// TIA Portal V17 export
// export: Created 2025-04-25T10:06:56.2061838Z, ExportSetting WithDefaults, DisplayName Totally Integrated Automation Portal, DisplayVersion V17 Update 8, DisplayName TIA Portal Openness, DisplayVersion V17 Update 8, DisplayName TIA Portal Version Control Interface, DisplayVersion V17, DisplayName SINAMICS Startdrive Advanced, DisplayVersion V17 SP2, DisplayName SINAMICS Startdrive G110M, G120, G120C, G120D, G120P, G115D, DisplayVersion V17 SP2, DisplayName SINAMICS Startdrive G130, G150, S120, S150, SINAMICS MV, S210, DisplayVersion V17 SP2, DisplayName STEP 7 Professional, DisplayVersion V17 Update 8, DisplayName SINUMERIK ONE STEP 7 Toolbox, DisplayVersion V17 Update 12, DisplayName SINUMERIK 840D sl STEP 7 Toolbox, DisplayVersion V17 Update 12, DisplayName STEP 7 Safety, DisplayVersion V17 Update 6, DisplayName WinCC Advanced / Unified PC, DisplayVersion V17 Update 8
FUNCTION "FC2810_U1_F4_GRIPPER" : Void   // FC2810, LAD
TITLE = FC2810_F4_GRIPPER
{ S7_Optimized_Access := 'FALSE' }
AUTHOR : ETXETAR
VERSION : 1.0
// stored: AutoNumber false, IsIECCheckEnabled false, SetENOAutomatically false, UDAEnableTagReadback false
   VAR_TEMP
      RET_VAL_1 : Int;
      UNIT_NUMBER : UInt;
      STATION_NUMBER : UInt;
   END_VAR
BEGIN

REGION Network 1: CALL FB2509 FIXTURE 1 GRIPPER
   // 2#0000_0001 OPTIONS 0 BIT 0 LOCATED INPUT 1 OPTION
   // 2#0000_0010 OPTIONS 0 BIT 1 LOCATED INPUT 2 OPTION
   // 2#0000_0100 OPTIONS 0 BIT 2 LOCATED INPUT 3 OPTION
   // 2#0000_1000 OPTIONS 0 BIT 3 LOCATED INPUT 4 OPTION
   // 2#0001_0000 OPTIONS 0 BIT 4 LOCATED PRESSURE INPUT 1 OPTION
   // 2#0010_0000 OPTIONS 0 BIT 5 LOCATED PRESSURE INPUT 2 OPTION
   // 2#0100_0000 OPTIONS 0 BIT 6 LOW PRESSURE INPUT 1 OPTION
   // 2#1000_0000 OPTIONS 0 BIT 7 SPARE OPTION
   // 
   // 2#0000_0001 OPTIONS 1 BIT 0 RETURNED INPUT 1 OPTION
   // 2#0000_0010 OPTIONS 1 BIT 1 RETURNED INPUT 2 OPTION
   // 2#0000_0100 OPTIONS 1 BIT 2 RETURNED INPUT 3 OPTION
   // 2#0000_1000 OPTIONS 1 BIT 3 RETURNED INPUT 4 OPTION
   // 2#0001_0000 OPTIONS 1 BIT 4 RETURNED PRESSURE INPUT 1 OPTION
   // 2#0010_0000 OPTIONS 1 BIT 5 RETURNED PRESSURE INPUT 2 OPTION
   // 2#0100_0000 OPTIONS 1 BIT 6 SPARE OPTION
   // 2#1000_0000 OPTIONS 1 BIT 7 SPARE OPTION
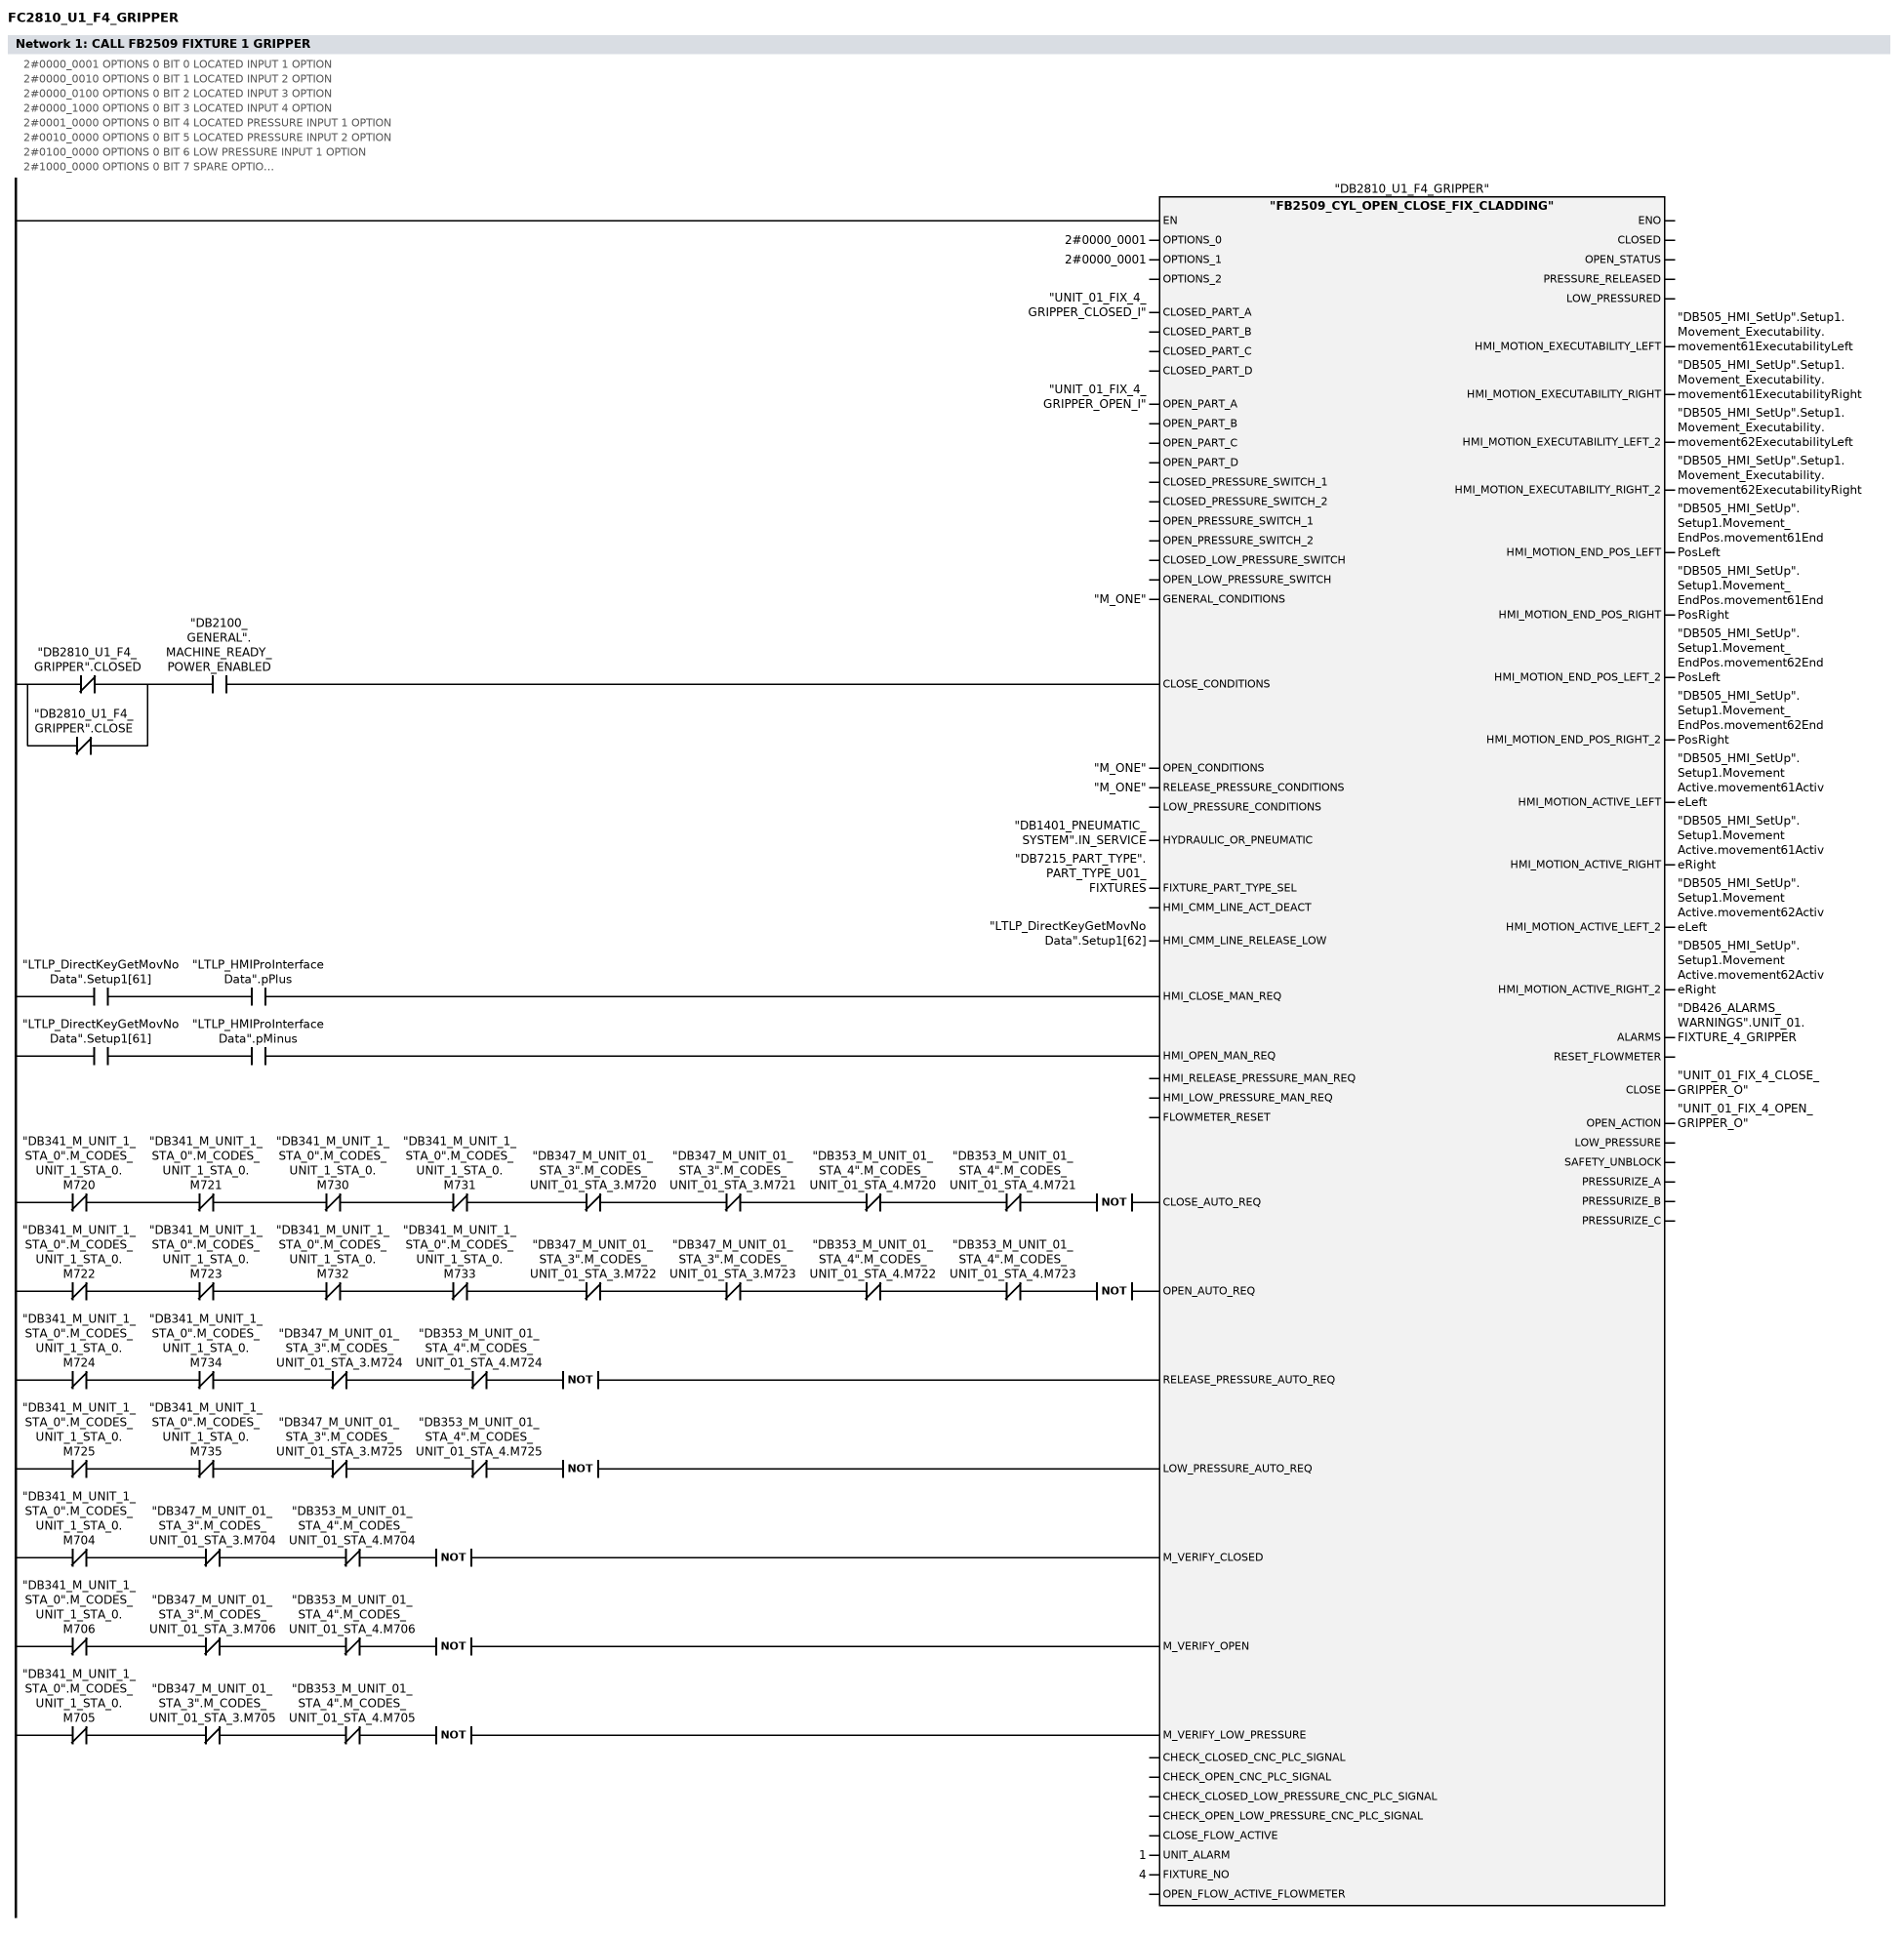
   RUNG wire#powerrail
      "DB2810_U1_F4_GRIPPER"(CLOSE_CONDITIONS := wire#w2, HMI_CLOSE_MAN_REQ := wire#w3, HMI_OPEN_MAN_REQ := wire#w4, CLOSE_AUTO_REQ := wire#w5, OPEN_AUTO_REQ := wire#w6, RELEASE_PRESSURE_AUTO_REQ := wire#w7, LOW_PRESSURE_AUTO_REQ := wire#w8, M_VERIFY_CLOSED := wire#w9, M_VERIFY_OPEN := wire#w10, M_VERIFY_LOW_PRESSURE := wire#w11, OPTIONS_0 := 2#0000_0001, OPTIONS_1 := 2#0000_0001, OPTIONS_2 :=, CLOSED_PART_A := "UNIT_01_FIX_4_GRIPPER_CLOSED_I", CLOSED_PART_B :=, CLOSED_PART_C :=, CLOSED_PART_D :=, OPEN_PART_A := "UNIT_01_FIX_4_GRIPPER_OPEN_I", OPEN_PART_B :=, OPEN_PART_C :=, OPEN_PART_D :=, CLOSED_PRESSURE_SWITCH_1 :=, CLOSED_PRESSURE_SWITCH_2 :=, OPEN_PRESSURE_SWITCH_1 :=, OPEN_PRESSURE_SWITCH_2 :=, CLOSED_LOW_PRESSURE_SWITCH :=, OPEN_LOW_PRESSURE_SWITCH :=, GENERAL_CONDITIONS := "M_ONE", OPEN_CONDITIONS := "M_ONE", RELEASE_PRESSURE_CONDITIONS := "M_ONE", LOW_PRESSURE_CONDITIONS :=, HYDRAULIC_OR_PNEUMATIC := "DB1401_PNEUMATIC_SYSTEM".IN_SERVICE, FIXTURE_PART_TYPE_SEL := "DB7215_PART_TYPE".PART_TYPE_U01_FIXTURES, HMI_CMM_LINE_ACT_DEACT :=, HMI_CMM_LINE_RELEASE_LOW := "LTLP_DirectKeyGetMovNoData".Setup1[62], HMI_RELEASE_PRESSURE_MAN_REQ :=, HMI_LOW_PRESSURE_MAN_REQ :=, FLOWMETER_RESET :=, CHECK_CLOSED_CNC_PLC_SIGNAL :=, CHECK_OPEN_CNC_PLC_SIGNAL :=, CHECK_CLOSED_LOW_PRESSURE_CNC_PLC_SIGNAL :=, CHECK_OPEN_LOW_PRESSURE_CNC_PLC_SIGNAL :=, CLOSE_FLOW_ACTIVE :=, UNIT_ALARM := 1, FIXTURE_NO := 4, OPEN_FLOW_ACTIVE_FLOWMETER :=, CLOSED =>, OPEN_STATUS =>, PRESSURE_RELEASED =>, LOW_PRESSURED =>, HMI_MOTION_EXECUTABILITY_LEFT => "DB505_HMI_SetUp".Setup1.Movement_Executability.movement61ExecutabilityLeft, HMI_MOTION_EXECUTABILITY_RIGHT => "DB505_HMI_SetUp".Setup1.Movement_Executability.movement61ExecutabilityRight, HMI_MOTION_EXECUTABILITY_LEFT_2 => "DB505_HMI_SetUp".Setup1.Movement_Executability.movement62ExecutabilityLeft, HMI_MOTION_EXECUTABILITY_RIGHT_2 => "DB505_HMI_SetUp".Setup1.Movement_Executability.movement62ExecutabilityRight, HMI_MOTION_END_POS_LEFT => "DB505_HMI_SetUp".Setup1.Movement_EndPos.movement61EndPosLeft, HMI_MOTION_END_POS_RIGHT => "DB505_HMI_SetUp".Setup1.Movement_EndPos.movement61EndPosRight, HMI_MOTION_END_POS_LEFT_2 => "DB505_HMI_SetUp".Setup1.Movement_EndPos.movement62EndPosLeft, HMI_MOTION_END_POS_RIGHT_2 => "DB505_HMI_SetUp".Setup1.Movement_EndPos.movement62EndPosRight, HMI_MOTION_ACTIVE_LEFT => "DB505_HMI_SetUp".Setup1.MovementActive.movement61ActiveLeft, HMI_MOTION_ACTIVE_RIGHT => "DB505_HMI_SetUp".Setup1.MovementActive.movement61ActiveRight, HMI_MOTION_ACTIVE_LEFT_2 => "DB505_HMI_SetUp".Setup1.MovementActive.movement62ActiveLeft, HMI_MOTION_ACTIVE_RIGHT_2 => "DB505_HMI_SetUp".Setup1.MovementActive.movement62ActiveRight, ALARMS => "DB426_ALARMS_WARNINGS".UNIT_01.FIXTURE_4_GRIPPER, RESET_FLOWMETER =>, CLOSE => "UNIT_01_FIX_4_CLOSE_GRIPPER_O", OPEN_ACTION => "UNIT_01_FIX_4_OPEN_GRIPPER_O", LOW_PRESSURE =>, SAFETY_UNBLOCK =>, PRESSURIZE_A =>, PRESSURIZE_B =>, PRESSURIZE_C =>)
   END_RUNG
   RUNG wire#powerrail
      I_Contact( "DB2810_U1_F4_GRIPPER".CLOSED )
      wire#w1
      Contact( "DB2100_GENERAL".MACHINE_READY_POWER_ENABLED )
   END_RUNG wire#w2
   RUNG wire#powerrail
      I_Contact( "DB2810_U1_F4_GRIPPER".CLOSE )
   END_RUNG wire#w1
   RUNG wire#powerrail
      Contact( "LTLP_DirectKeyGetMovNoData".Setup1[61] )
      Contact( "LTLP_HMIProInterfaceData".pPlus )
   END_RUNG wire#w3
   RUNG wire#powerrail
      Contact( "LTLP_DirectKeyGetMovNoData".Setup1[61] )
      Contact( "LTLP_HMIProInterfaceData".pMinus )
   END_RUNG wire#w4
   RUNG wire#powerrail
      I_Contact( "DB341_M_UNIT_1_STA_0".M_CODES_UNIT_1_STA_0.M720 )
      I_Contact( "DB341_M_UNIT_1_STA_0".M_CODES_UNIT_1_STA_0.M721 )
      I_Contact( "DB341_M_UNIT_1_STA_0".M_CODES_UNIT_1_STA_0.M730 )
      I_Contact( "DB341_M_UNIT_1_STA_0".M_CODES_UNIT_1_STA_0.M731 )
      I_Contact( "DB347_M_UNIT_01_STA_3".M_CODES_UNIT_01_STA_3.M720 )
      I_Contact( "DB347_M_UNIT_01_STA_3".M_CODES_UNIT_01_STA_3.M721 )
      I_Contact( "DB353_M_UNIT_01_STA_4".M_CODES_UNIT_01_STA_4.M720 )
      I_Contact( "DB353_M_UNIT_01_STA_4".M_CODES_UNIT_01_STA_4.M721 )
      Not()
   END_RUNG wire#w5
   RUNG wire#powerrail
      I_Contact( "DB341_M_UNIT_1_STA_0".M_CODES_UNIT_1_STA_0.M722 )
      I_Contact( "DB341_M_UNIT_1_STA_0".M_CODES_UNIT_1_STA_0.M723 )
      I_Contact( "DB341_M_UNIT_1_STA_0".M_CODES_UNIT_1_STA_0.M732 )
      I_Contact( "DB341_M_UNIT_1_STA_0".M_CODES_UNIT_1_STA_0.M733 )
      I_Contact( "DB347_M_UNIT_01_STA_3".M_CODES_UNIT_01_STA_3.M722 )
      I_Contact( "DB347_M_UNIT_01_STA_3".M_CODES_UNIT_01_STA_3.M723 )
      I_Contact( "DB353_M_UNIT_01_STA_4".M_CODES_UNIT_01_STA_4.M722 )
      I_Contact( "DB353_M_UNIT_01_STA_4".M_CODES_UNIT_01_STA_4.M723 )
      Not()
   END_RUNG wire#w6
   RUNG wire#powerrail
      I_Contact( "DB341_M_UNIT_1_STA_0".M_CODES_UNIT_1_STA_0.M724 )
      I_Contact( "DB341_M_UNIT_1_STA_0".M_CODES_UNIT_1_STA_0.M734 )
      I_Contact( "DB347_M_UNIT_01_STA_3".M_CODES_UNIT_01_STA_3.M724 )
      I_Contact( "DB353_M_UNIT_01_STA_4".M_CODES_UNIT_01_STA_4.M724 )
      Not()
   END_RUNG wire#w7
   RUNG wire#powerrail
      I_Contact( "DB341_M_UNIT_1_STA_0".M_CODES_UNIT_1_STA_0.M725 )
      I_Contact( "DB341_M_UNIT_1_STA_0".M_CODES_UNIT_1_STA_0.M735 )
      I_Contact( "DB347_M_UNIT_01_STA_3".M_CODES_UNIT_01_STA_3.M725 )
      I_Contact( "DB353_M_UNIT_01_STA_4".M_CODES_UNIT_01_STA_4.M725 )
      Not()
   END_RUNG wire#w8
   RUNG wire#powerrail
      I_Contact( "DB341_M_UNIT_1_STA_0".M_CODES_UNIT_1_STA_0.M704 )
      I_Contact( "DB347_M_UNIT_01_STA_3".M_CODES_UNIT_01_STA_3.M704 )
      I_Contact( "DB353_M_UNIT_01_STA_4".M_CODES_UNIT_01_STA_4.M704 )
      Not()
   END_RUNG wire#w9
   RUNG wire#powerrail
      I_Contact( "DB341_M_UNIT_1_STA_0".M_CODES_UNIT_1_STA_0.M706 )
      I_Contact( "DB347_M_UNIT_01_STA_3".M_CODES_UNIT_01_STA_3.M706 )
      I_Contact( "DB353_M_UNIT_01_STA_4".M_CODES_UNIT_01_STA_4.M706 )
      Not()
   END_RUNG wire#w10
   RUNG wire#powerrail
      I_Contact( "DB341_M_UNIT_1_STA_0".M_CODES_UNIT_1_STA_0.M705 )
      I_Contact( "DB347_M_UNIT_01_STA_3".M_CODES_UNIT_01_STA_3.M705 )
      I_Contact( "DB353_M_UNIT_01_STA_4".M_CODES_UNIT_01_STA_4.M705 )
      Not()
   END_RUNG wire#w11
   // the same network as SCL:
   "DB2810_U1_F4_GRIPPER"(OPTIONS_0 := 2#0000_0001,   // "FB2509_CYL_OPEN_CLOSE_FIX_CLADDING"
                          OPTIONS_1 := 2#0000_0001,
                          CLOSED_PART_A := "UNIT_01_FIX_4_GRIPPER_CLOSED_I",
                          OPEN_PART_A := "UNIT_01_FIX_4_GRIPPER_OPEN_I",
                          GENERAL_CONDITIONS := "M_ONE",
                          CLOSE_CONDITIONS := (NOT "DB2810_U1_F4_GRIPPER".CLOSED OR NOT "DB2810_U1_F4_GRIPPER".CLOSE) AND "DB2100_GENERAL".MACHINE_READY_POWER_ENABLED,
                          OPEN_CONDITIONS := "M_ONE",
                          RELEASE_PRESSURE_CONDITIONS := "M_ONE",
                          HYDRAULIC_OR_PNEUMATIC := "DB1401_PNEUMATIC_SYSTEM".IN_SERVICE,
                          FIXTURE_PART_TYPE_SEL := "DB7215_PART_TYPE".PART_TYPE_U01_FIXTURES,
                          HMI_CMM_LINE_RELEASE_LOW := "LTLP_DirectKeyGetMovNoData".Setup1[62],
                          HMI_CLOSE_MAN_REQ := "LTLP_DirectKeyGetMovNoData".Setup1[61] AND "LTLP_HMIProInterfaceData".pPlus,
                          HMI_OPEN_MAN_REQ := "LTLP_DirectKeyGetMovNoData".Setup1[61] AND "LTLP_HMIProInterfaceData".pMinus,
                          CLOSE_AUTO_REQ := NOT (NOT "DB341_M_UNIT_1_STA_0".M_CODES_UNIT_1_STA_0.M720 AND NOT "DB341_M_UNIT_1_STA_0".M_CODES_UNIT_1_STA_0.M721 AND NOT "DB341_M_UNIT_1_STA_0".M_CODES_UNIT_1_STA_0.M730 AND NOT "DB341_M_UNIT_1_STA_0".M_CODES_UNIT_1_STA_0.M731 AND NOT "DB347_M_UNIT_01_STA_3".M_CODES_UNIT_01_STA_3.M720 AND NOT "DB347_M_UNIT_01_STA_3".M_CODES_UNIT_01_STA_3.M721 AND NOT "DB353_M_UNIT_01_STA_4".M_CODES_UNIT_01_STA_4.M720 AND NOT "DB353_M_UNIT_01_STA_4".M_CODES_UNIT_01_STA_4.M721),
                          OPEN_AUTO_REQ := NOT (NOT "DB341_M_UNIT_1_STA_0".M_CODES_UNIT_1_STA_0.M722 AND NOT "DB341_M_UNIT_1_STA_0".M_CODES_UNIT_1_STA_0.M723 AND NOT "DB341_M_UNIT_1_STA_0".M_CODES_UNIT_1_STA_0.M732 AND NOT "DB341_M_UNIT_1_STA_0".M_CODES_UNIT_1_STA_0.M733 AND NOT "DB347_M_UNIT_01_STA_3".M_CODES_UNIT_01_STA_3.M722 AND NOT "DB347_M_UNIT_01_STA_3".M_CODES_UNIT_01_STA_3.M723 AND NOT "DB353_M_UNIT_01_STA_4".M_CODES_UNIT_01_STA_4.M722 AND NOT "DB353_M_UNIT_01_STA_4".M_CODES_UNIT_01_STA_4.M723),
                          RELEASE_PRESSURE_AUTO_REQ := NOT (NOT "DB341_M_UNIT_1_STA_0".M_CODES_UNIT_1_STA_0.M724 AND NOT "DB341_M_UNIT_1_STA_0".M_CODES_UNIT_1_STA_0.M734 AND NOT "DB347_M_UNIT_01_STA_3".M_CODES_UNIT_01_STA_3.M724 AND NOT "DB353_M_UNIT_01_STA_4".M_CODES_UNIT_01_STA_4.M724),
                          LOW_PRESSURE_AUTO_REQ := NOT (NOT "DB341_M_UNIT_1_STA_0".M_CODES_UNIT_1_STA_0.M725 AND NOT "DB341_M_UNIT_1_STA_0".M_CODES_UNIT_1_STA_0.M735 AND NOT "DB347_M_UNIT_01_STA_3".M_CODES_UNIT_01_STA_3.M725 AND NOT "DB353_M_UNIT_01_STA_4".M_CODES_UNIT_01_STA_4.M725),
                          M_VERIFY_CLOSED := NOT (NOT "DB341_M_UNIT_1_STA_0".M_CODES_UNIT_1_STA_0.M704 AND NOT "DB347_M_UNIT_01_STA_3".M_CODES_UNIT_01_STA_3.M704 AND NOT "DB353_M_UNIT_01_STA_4".M_CODES_UNIT_01_STA_4.M704),
                          M_VERIFY_OPEN := NOT (NOT "DB341_M_UNIT_1_STA_0".M_CODES_UNIT_1_STA_0.M706 AND NOT "DB347_M_UNIT_01_STA_3".M_CODES_UNIT_01_STA_3.M706 AND NOT "DB353_M_UNIT_01_STA_4".M_CODES_UNIT_01_STA_4.M706),
                          M_VERIFY_LOW_PRESSURE := NOT (NOT "DB341_M_UNIT_1_STA_0".M_CODES_UNIT_1_STA_0.M705 AND NOT "DB347_M_UNIT_01_STA_3".M_CODES_UNIT_01_STA_3.M705 AND NOT "DB353_M_UNIT_01_STA_4".M_CODES_UNIT_01_STA_4.M705),
                          UNIT_ALARM := 1,
                          FIXTURE_NO := 4,
                          HMI_MOTION_EXECUTABILITY_LEFT => "DB505_HMI_SetUp".Setup1.Movement_Executability.movement61ExecutabilityLeft,
                          HMI_MOTION_EXECUTABILITY_RIGHT => "DB505_HMI_SetUp".Setup1.Movement_Executability.movement61ExecutabilityRight,
                          HMI_MOTION_EXECUTABILITY_LEFT_2 => "DB505_HMI_SetUp".Setup1.Movement_Executability.movement62ExecutabilityLeft,
                          HMI_MOTION_EXECUTABILITY_RIGHT_2 => "DB505_HMI_SetUp".Setup1.Movement_Executability.movement62ExecutabilityRight,
                          HMI_MOTION_END_POS_LEFT => "DB505_HMI_SetUp".Setup1.Movement_EndPos.movement61EndPosLeft,
                          HMI_MOTION_END_POS_RIGHT => "DB505_HMI_SetUp".Setup1.Movement_EndPos.movement61EndPosRight,
                          HMI_MOTION_END_POS_LEFT_2 => "DB505_HMI_SetUp".Setup1.Movement_EndPos.movement62EndPosLeft,
                          HMI_MOTION_END_POS_RIGHT_2 => "DB505_HMI_SetUp".Setup1.Movement_EndPos.movement62EndPosRight,
                          HMI_MOTION_ACTIVE_LEFT => "DB505_HMI_SetUp".Setup1.MovementActive.movement61ActiveLeft,
                          HMI_MOTION_ACTIVE_RIGHT => "DB505_HMI_SetUp".Setup1.MovementActive.movement61ActiveRight,
                          HMI_MOTION_ACTIVE_LEFT_2 => "DB505_HMI_SetUp".Setup1.MovementActive.movement62ActiveLeft,
                          HMI_MOTION_ACTIVE_RIGHT_2 => "DB505_HMI_SetUp".Setup1.MovementActive.movement62ActiveRight,
                          ALARMS => "DB426_ALARMS_WARNINGS".UNIT_01.FIXTURE_4_GRIPPER,
                          CLOSE => "UNIT_01_FIX_4_CLOSE_GRIPPER_O",
                          OPEN_ACTION => "UNIT_01_FIX_4_OPEN_GRIPPER_O");
END_REGION
END_FUNCTION
